INTERFACE I_Enablable EXTENDS I_Base

METHOD Disable
VAR_INPUT
END_VAR
END_METHOD

METHOD Enable
VAR_INPUT
END_VAR
END_METHOD

{attribute 'monitoring' := 'call'}
PROPERTY Enabled : BOOL
GET
END_GET
END_PROPERTY

END_INTERFACE

(* stored: Version 1.1.0.1, ProductVersion 3.1.4026.18
   Itf I_Enablable: Id {30dac2a0-3727-432e-9194-a136d2a3adb1}
   Method Disable: Id {a3bfae26-51d5-4c76-8cc5-0002149fcd5d}
   Method Enable: Id {53da13cd-3792-4478-b0f3-a241954ca654}
   Property Enabled: Id {be153cdf-28f3-4091-a3c0-53a071f3041a}
   Get Get: Id {e5f85cb6-404e-4661-87f1-a314c8a52af3} *)
